(* Logix 5000 project; controller Commerford_topping_5477_V3 vendor 1 type 14 code 222 rev 33.11; software revision 33.02 *)

TASK MainTask (continuous, watchdog 500 ms) : MainProgram
TASK SafetyTask (periodic, rate 20 ms, priority 10, watchdog 20 ms, safety) : SafetyProgram
TASK Unit6_Topping_system (event, rate 10 ms, priority 10, watchdog 500 ms) : UN6_Object, UN6_EM1_Buffertank, UN6_EM2_Color_1, UN6_EM3_Color_2, UN6_EM4_Color_3, UN6_EM5_No_Color

MODULES
   Local : vendor 1 type 14 code 222 (5069 0, rev 33.11)
END_MODULES

TYPE Descriptor :   // is used for recipes
STRUCT
   Value : REAL;   // Parameter Values
END_STRUCT
END_TYPE

TYPE EquipmentModule :   // EquipmentModule
STRUCT
   Selected : BOOL;   // EquipmentModule is active
   State_in : DINT;   // EM State request
   State_out : DINT;   // EM State complete
   Current_Action : STRING_32;   // Contains information about current action of equipment module
   Force_Stop : BOOL;   // Sets the statemodel to Stopping
   Force_Abort : BOOL;   // Sets the statemodel to Aborting
   Suspend_Trigger : BOOL;   // Requests a Suspending state
   Reset_Signal : BOOL;   // Reset for entire EM, this will be done by 1. Resetting 2. Clearing 3. HMI_Reset
   Faulted : BOOL;   // EquipmentModule is faulted locally
   CM_Force_Stop : BOOL;   // Sets the statemodel to Stopping, ONLY USED BY CM AOI. DO NOT USE OTHERWISE!!
   CM_Force_Abort : BOOL;   // Sets the statemodel to Aborting, ONLY USED BY CM AOI. DO NOT USE OTHERWISE!!
   _SEQ : EquipmentModule_SEQ;
END_STRUCT
END_TYPE

TYPE EquipmentModule_SEQ :
STRUCT
   Clearing : INT;   // Step nummer
   Activating : INT;   // Step nummer
   Deactivating : INT;   // Step nummer
   Aborting : INT;   // Step nummer
   Resetting : INT;   // Step nummer
END_STRUCT
END_TYPE

TYPE MasterRecipeSelect :
STRUCT
   Recipe : STRING_476;
   SelectedRecipeNum : DINT;
   SelectedProces : DINT;
   RunRecipe : BOOL;   // Set to true to download recipe to proces
   Process : STRING_476;
END_STRUCT
END_TYPE

TYPE Packml_States :   // Enum for packml states
STRUCT
   Aborting : BOOL;   // Packml state
   Aborted : BOOL;   // Packml state
   Clearing : BOOL;   // Packml state
   Stopping : BOOL;   // Packml state
   Stopped : BOOL;   // Packml state
   Resetting : BOOL;   // Packml state
   Idle : BOOL;   // Packml state
   Starting : BOOL;   // Packml state
   Execute : BOOL;   // Packml state
   Holding : BOOL;   // Packml state
   Held : BOOL;   // Packml state
   Unholding : BOOL;   // Packml state
   Suspending : BOOL;   // Packml state
   Suspended : BOOL;   // Packml state
   Unsuspending : BOOL;   // Packml state
   Completing : BOOL;   // Packml state
   Complete : BOOL;   // Packml state
END_STRUCT
END_TYPE

TYPE PLMs :   // Status tags are used to describe the operation of the unit machine. Status tags include state commands which describe the state transitions in the Base State Model. The status tags also include parameters and process variables which describe how the machine operates.
STRUCT
   UnitModeCurrent : DINT;   // Unit Mode in Current Use
   UnitModeRequested : BOOL;   // Requested Unit Mode Change
   UnitModeChangeInProcess : BOOL;   // Requested Unit Mode Change in Process
   StateCurrent : DINT;   // Current State Number
   StateRequested : DINT;   // Target State.
   StateChangeInProcess : BOOL;   // State Change in Process.
   MachSpeed : REAL;   // Current Machine Speed
   CurMachSpeed : REAL;   // Current Machine Speed in Primary Packages/Minute
   MaterialInterlock : BOOL;   // Materials Ready
   UnitFaulted : BOOL;   // Machine is faulted
END_STRUCT
END_TYPE

TYPE PMLc :   // Command tags are used to control the operation of the unit machine. Command tags include unit state commands which control the state transitions in the Base State Model.
STRUCT
   UnitMode : DINT;   // This value is predefined by the user/OEM, and are the desired unit modes of the machine.
   UnitModeChangeRequest : BOOL;   // When a unit mode request takes place a numerical value must be present in the Command.UnitMode tag to change the unit mode.
   MaterialsInterlocks : BOOL;
   CntrlCmd : DINT;   // 0 Undefined 1 Reset 2 Start 3 Stop 4 Hold 5 Unhold 6 Suspend 7 Unsuspend 8 Abort 9 Clear
   CmdChangeRequest : BOOL;   // This CmdChangeRequest bit will command the machine to proceed to change the state to the target state. The tag can be used to condition when a change of state can occur. The target state will be one of the states in the base state model.
END_STRUCT
END_TYPE

TYPE Process_Status :
STRUCT
   Running : BOOL;   // Phase is executing Running logic
   Complete : BOOL;   // Phase is completed, waiting for reset command
   Held : BOOL;   // Phase is held, waiting for Restart command
   Idle : BOOL;   // Phase is Idle, waiting for Start command
   Resetting : BOOL;   // Phase is executing Resetting logic
   Stopped : BOOL;   // Phase is Stopped, waiting for Reset command
   Aborted : BOOL;   // Phase is Aborted, waiting for Reset command
   Aborting : BOOL;   // Phase is executing Aborting logic
   Stopping : BOOL;   // Phase is executing Stopping logic
   Holding : BOOL;   // Phase is executing Holding logic
   Restarting : BOOL;   // Phase is executing Restarting logic
   Ready : BOOL;   // Phase Completed, phase is ready to recieve new commands
END_STRUCT
END_TYPE

TYPE ProcessModule :
STRUCT
   Selected : BOOL;   // Process is active
   State_in : DINT;   // Process State request
   State_out : DINT;   // Process State complete
   Force_Stop : BOOL;   // Sets the statemodel to Stopping
   Force_Abort : BOOL;   // Sets the statemodel to Aborting
   Suspend_Trigger : BOOL;   // Requests a Suspending state
   Faulted : BOOL;   // Process is faulted locally
   Status : Process_Status;   // Status of process
END_STRUCT
END_TYPE

TYPE StateCurrentTime_array :   // sub array
STRUCT
   Mode : DINT[18];
END_STRUCT
END_TYPE

TYPE STRING_476 :   // Max chars HMI supports.
STRUCT
   LEN : DINT;
   DATA : SINT[476];
END_STRUCT
END_TYPE

ADD_ON_INSTRUCTION EquipmentModule_Link   (* revision 1.1, vendor WPI *)
// Revision note:
// 1.1 - CM faults reset
VAR_IN_OUT
   PackML : ISA_TR_88_00_02; {required}
   EquipmentModule : EquipmentModule; {required}
   bStateTransitions : DINT[32]; {required}
END_VAR
VAR_INPUT
   EM_ID : DINT; {required}
   Select : BOOL; {visible}   // Selecting EM will incuding in Unit state transitions
END_VAR
VAR_OUTPUT
   Sts_EM_Selected : BOOL; {access Read Only, visible}
   OwnershipFault : BOOL; {access Read Only, visible}
   Sts_Clearing_PC : BOOL; {access Read Only, visible}
   Sts_Starting_PC : BOOL; {access Read Only, visible}
   Sts_Executing : BOOL; {access Read Only, visible}
   Sts_Stopping_PC : BOOL; {access Read Only, visible}
   Sts_Aborting_PC : BOOL; {access Read Only, visible}
   Sts_Holding_PC : BOOL; {access Read Only, visible}
   Sts_Unholding_PC : BOOL; {access Read Only, visible}
   Sts_Suspending_PC : BOOL; {access Read Only, visible}
   Sts_Resetting_PC : BOOL; {access Read Only, visible}
   Sts_Unsuspending_PC : BOOL; {access Read Only, visible}
   Sts_Completing_PC : BOOL; {access Read Only, visible}
   Sts_SuspendTrigger : BOOL; {access Read Only, visible}
   Sts_Faulted : BOOL; {access Read Only, visible}
   Sts_Force_Stop : BOOL; {access Read Only, visible}
   Sts_Force_Abort : BOOL; {access Read Only, visible}
END_VAR
VAR
   AsignOwnership : BOOL; {access None}
   UnasignOwnership : BOOL; {access None}
END_VAR

ROUTINE Logic   (* ladder *)
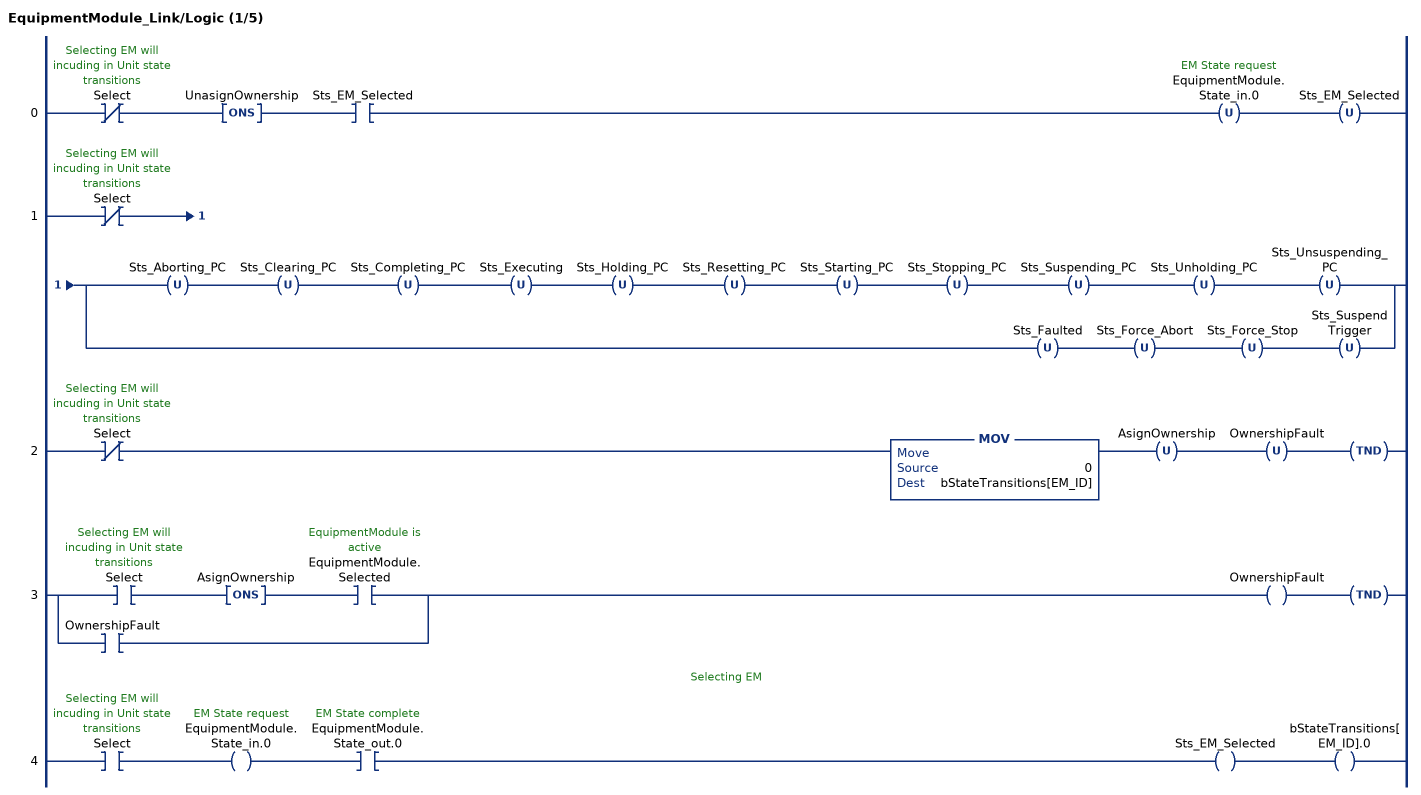
   0: XIO(Select)ONS(UnasignOwnership)XIC(Sts_EM_Selected)OTU(EquipmentModule.State_in.0)OTU(Sts_EM_Selected);
   1: XIO(Select)[OTU(Sts_Aborting_PC) OTU(Sts_Clearing_PC) OTU(Sts_Completing_PC) OTU(Sts_Executing) OTU(Sts_Holding_PC) OTU(Sts_Resetting_PC) OTU(Sts_Starting_PC) OTU(Sts_Stopping_PC) OTU(Sts_Suspending_PC) OTU(Sts_Unholding_PC) OTU(Sts_Unsuspending_PC) ,OTU(Sts_Faulted) OTU(Sts_Force_Abort) OTU(Sts_Force_Stop) OTU(Sts_SuspendTrigger) ];
   2: XIO(Select)MOV(0,bStateTransitions[EM_ID])OTU(AsignOwnership)OTU(OwnershipFault)TND();
   3: [XIC(Select) ONS(AsignOwnership) XIC(EquipmentModule.Selected) ,XIC(OwnershipFault) ]OTE(OwnershipFault)TND();
   // Selecting EM
   4: XIC(Select)OTE(EquipmentModule.State_in.0)XIC(EquipmentModule.State_out.0)OTE(Sts_EM_Selected)OTE(bStateTransitions[EM_ID].0);
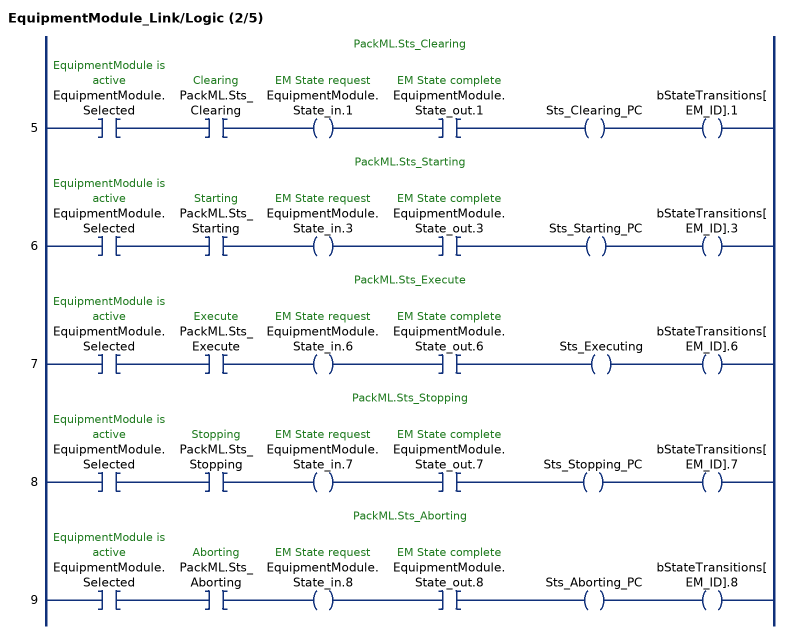
   // PackML.Sts_Clearing
   5: XIC(EquipmentModule.Selected)XIC(PackML.Sts_Clearing)OTE(EquipmentModule.State_in.1)XIC(EquipmentModule.State_out.1)OTE(Sts_Clearing_PC)OTE(bStateTransitions[EM_ID].1);
   // PackML.Sts_Starting
   6: XIC(EquipmentModule.Selected)XIC(PackML.Sts_Starting)OTE(EquipmentModule.State_in.3)XIC(EquipmentModule.State_out.3)OTE(Sts_Starting_PC)OTE(bStateTransitions[EM_ID].3);
   // PackML.Sts_Execute
   7: XIC(EquipmentModule.Selected)XIC(PackML.Sts_Execute)OTE(EquipmentModule.State_in.6)XIC(EquipmentModule.State_out.6)OTE(Sts_Executing)OTE(bStateTransitions[EM_ID].6);
   // PackML.Sts_Stopping
   8: XIC(EquipmentModule.Selected)XIC(PackML.Sts_Stopping)OTE(EquipmentModule.State_in.7)XIC(EquipmentModule.State_out.7)OTE(Sts_Stopping_PC)OTE(bStateTransitions[EM_ID].7);
   // PackML.Sts_Aborting
   9: XIC(EquipmentModule.Selected)XIC(PackML.Sts_Aborting)OTE(EquipmentModule.State_in.8)XIC(EquipmentModule.State_out.8)OTE(Sts_Aborting_PC)OTE(bStateTransitions[EM_ID].8);
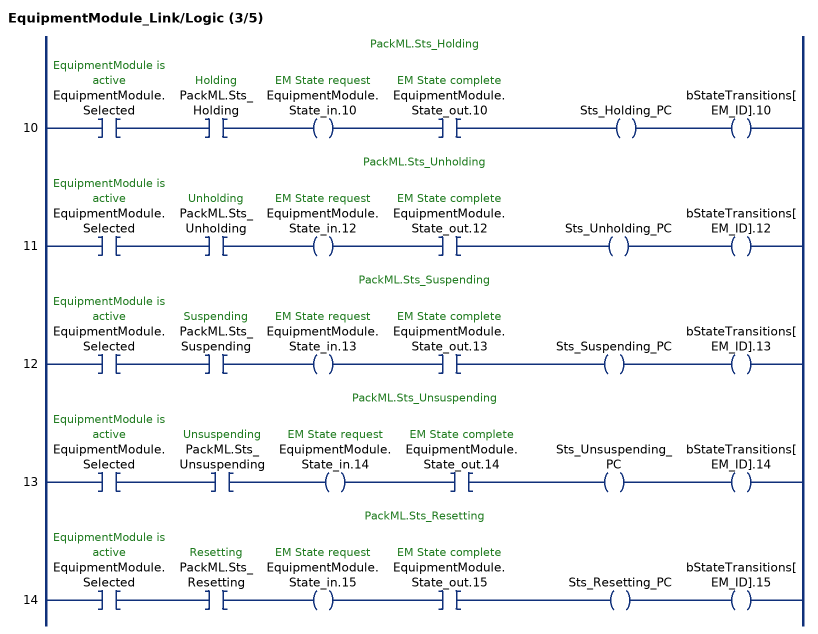
   // PackML.Sts_Holding
   10: XIC(EquipmentModule.Selected)XIC(PackML.Sts_Holding)OTE(EquipmentModule.State_in.10)XIC(EquipmentModule.State_out.10)OTE(Sts_Holding_PC)OTE(bStateTransitions[EM_ID].10);
   // PackML.Sts_Unholding
   11: XIC(EquipmentModule.Selected)XIC(PackML.Sts_Unholding)OTE(EquipmentModule.State_in.12)XIC(EquipmentModule.State_out.12)OTE(Sts_Unholding_PC)OTE(bStateTransitions[EM_ID].12);
   // PackML.Sts_Suspending
   12: XIC(EquipmentModule.Selected)XIC(PackML.Sts_Suspending)OTE(EquipmentModule.State_in.13)XIC(EquipmentModule.State_out.13)OTE(Sts_Suspending_PC)OTE(bStateTransitions[EM_ID].13);
   // PackML.Sts_Unsuspending
   13: XIC(EquipmentModule.Selected)XIC(PackML.Sts_Unsuspending)OTE(EquipmentModule.State_in.14)XIC(EquipmentModule.State_out.14)OTE(Sts_Unsuspending_PC)OTE(bStateTransitions[EM_ID].14);
   // PackML.Sts_Resetting
   14: XIC(EquipmentModule.Selected)XIC(PackML.Sts_Resetting)OTE(EquipmentModule.State_in.15)XIC(EquipmentModule.State_out.15)OTE(Sts_Resetting_PC)OTE(bStateTransitions[EM_ID].15);
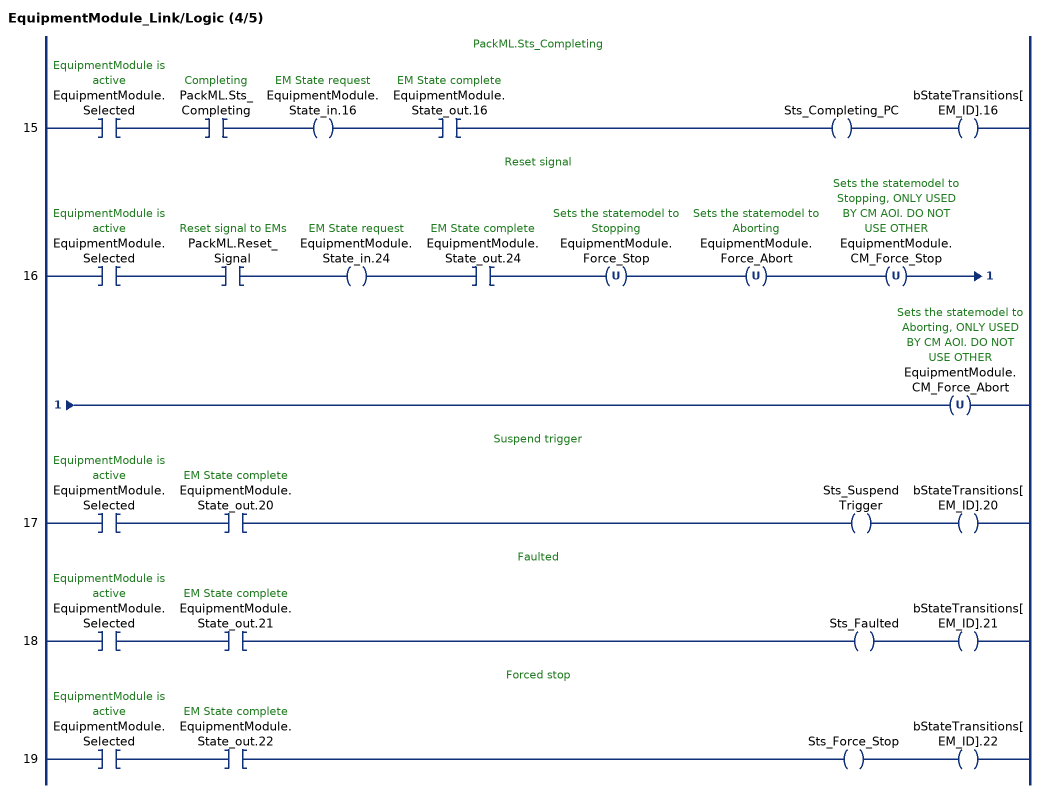
   // PackML.Sts_Completing
   15: XIC(EquipmentModule.Selected)XIC(PackML.Sts_Completing)OTE(EquipmentModule.State_in.16)XIC(EquipmentModule.State_out.16)OTE(Sts_Completing_PC)OTE(bStateTransitions[EM_ID].16);
   // Reset signal
   16: XIC(EquipmentModule.Selected)XIC(PackML.Reset_Signal)OTE(EquipmentModule.State_in.24)XIC(EquipmentModule.State_out.24)OTU(EquipmentModule.Force_Stop)OTU(EquipmentModule.Force_Abort)OTU(EquipmentModule.CM_Force_Stop)OTU(EquipmentModule.CM_Force_Abort);
   // Suspend trigger
   17: XIC(EquipmentModule.Selected)XIC(EquipmentModule.State_out.20)OTE(Sts_SuspendTrigger)OTE(bStateTransitions[EM_ID].20);
   // Faulted
   18: XIC(EquipmentModule.Selected)XIC(EquipmentModule.State_out.21)OTE(Sts_Faulted)OTE(bStateTransitions[EM_ID].21);
   // Forced stop
   19: XIC(EquipmentModule.Selected)XIC(EquipmentModule.State_out.22)OTE(Sts_Force_Stop)OTE(bStateTransitions[EM_ID].22);
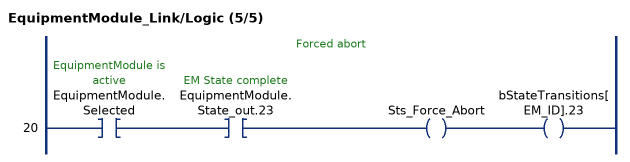
   // Forced abort
   20: XIC(EquipmentModule.Selected)XIC(EquipmentModule.State_out.23)OTE(Sts_Force_Abort)OTE(bStateTransitions[EM_ID].23);
END_ROUTINE
END_ADD_ON_INSTRUCTION

ADD_ON_INSTRUCTION ISA_TR_88_00_02   (* revision 1.2, ExecutePrescan *)
// Machine and Unit States:
// An Implementation Example of
// ISA-88
// Revision note:
// Processactive update
// Help:
// Read parameter list for documentation
VAR_IN_OUT
   PackTags : PACKMLv30; {required}
   EquipmentModules : DINT[32]; {required}
END_VAR
VAR_OUTPUT
   Sts_SC_Status : UDINT; {access Read Only, visible}
   Sts_Clearing : BOOL; {access Read Only, visible}   // Clearing
   Sts_Stopped : BOOL; {access Read Only, visible}   // Stopped
   Sts_Starting : BOOL; {access Read Only, visible}   // Starting
   Sts_Idle : BOOL; {access Read Only, visible}   // Idle
   Sts_Suspended : BOOL; {access Read Only, visible}   // Suspended
   Sts_Execute : BOOL; {access Read Only, visible}   // Execute
   Sts_Stopping : BOOL; {access Read Only, visible}   // Stopping
   Sts_Aborting : BOOL; {access Read Only, visible}   // Aborting
   Sts_Aborted : BOOL; {access Read Only, visible}   // Aborted
   Sts_Holding : BOOL; {access Read Only, visible}   // Holding
   Sts_Held : BOOL; {access Read Only, visible}   // Held
   Sts_Unholding : BOOL; {access Read Only, visible}   // Unholding
   Sts_Suspending : BOOL; {access Read Only, visible}   // Suspending
   Sts_Unsuspending : BOOL; {access Read Only, visible}   // Unsuspending
   Sts_Resetting : BOOL; {access Read Only, visible}   // Resetting
   Sts_Completing : BOOL; {access Read Only, visible}   // Completing
   Sts_Complete : BOOL; {access Read Only, visible}   // Complete
   Sts_Automatic : BOOL; {access Read Only, visible}   // Machine is in fully automatic mode
   Sts_Maintenance : BOOL; {access Read Only, visible}   // Machine is in Maintenance
   Sts_Manual : BOOL; {access Read Only, visible}   // Machine is in Manual
END_VAR
VAR_INPUT
   Process_Selected : SINT; {visible}   // Recipe number selects which PackTag.command.product[#] will be used.
END_VAR
VAR_OUTPUT
   Sts_MachineFaulted : BOOL; {access Read Only, visible}   // Machine recieved an fault trigger
END_VAR
VAR_INPUT
   HMI_Reset : BOOL;   // Common reset for all EMs
END_VAR
VAR_OUTPUT
   Sts_ProcessActive : BOOL; {access Read Only, visible}   // Machine is running a process.
   Reset_Signal : BOOL; {access Read Only}   // Reset signal to EMs
END_VAR
VAR_IN_OUT
   Processes : DINT[32]; {required}
   Cnf_EnableMachineStates : Packml_States; {required}
END_VAR
VAR
   MachineState : USINT := 255; {access None}   // Technical Report Equipment States: 1 Clearing 2 Stopped 3 Starting 4 Idle 5 Suspended 6 Execute 7 Stopping 8 Aborting 9 Aborted 10 Holding 11 Held 12 Unholding 13 Suspending 14 Unsuspending 15 Resetting 16 Completing 17 Complete
   wrk_compare_UDINT : UDINT := 65535; {access None}
   wrk_Aborting_to_Aborted : UDINT := 2#0000_0000_0000_0000_1111_1111_1111_1111; {access None}
   i : DINT; {access None}   // index num, only for local use. used for forloops
   Wrk_Aborting_to_Aborted_PC : BOOL; {access None}   // EquipmentModule(s) Aborting_to_Aborted Proces Complete
   FALSE : BOOL; {access None}   // always false
   TRUE : BOOL; {access None}   // always true
   wrk_Conversion : DINT; {access None}
   temp_sum : DINT; {access None}   // local storage
   wrk_Stopping_to_Stopped : UDINT; {access None}
   wrk_Starting_to_Execute : UDINT; {access None}
   wrk_Clearing_to_Stopped : UDINT; {access None}
   wrk_Holding_to_Held : UDINT; {access None}
   wrk_Unholding_to_Execute : UDINT; {access None}
   wrk_Suspending_to_Suspended : UDINT; {access None}
   wrk_Unsuspending_to_Execute : UDINT; {access None}
   wrk_Resetting_to_Idle : UDINT; {access None}
   wrk_Completing_to_Completed : UDINT; {access None}
   wrk_prev_state : DINT; {access None}   // local mem
   MachineMode : DINT; {access None}
   wrk_SwitchLayer_To_Maintenance : DINT; {access None}
   wrk_SwitchLayer_To_Manual : DINT; {access None}
   wrk_SwitchLayer_To_Automatic : DINT; {access None}
   k : DINT; {access None}   // nested index num
   ArraySize : DINT[5]; {access None}   // local array size
   wrk_RecipeNumber : DINT; {access None}   // local RecipeNum
   DEL_T_Refresh_PackTag_Status : FBD_TIMER; {access None}
   T_second_puls : FBD_TIMER; {access None}   // local timer for just 1 second
   T_Refresh_PackTag_Administration : FBD_TIMER; {access None}   // local timer
   wrk_DateTime : LINT; {access None}
   wrk_Execute_to_Completing : UDINT; {access None}
   T_ResetSignal_ON : FBD_TIMER; {access None}   // Local reset timer
   T_ResetSignal_OFF : FBD_TIMER; {access None}   // local reset timer
   T_ResetSignal_HMI : FBD_TIMER; {access None}   // reset timer from HMI
   StateHistory : StateHistory[10]; {access Read Only}
   debugProg : DINT; {access None}
   wrk_HandHalt : BOOL; {access None}   // machine is forced to stop by user
   Wrk_EM_Restting : UDINT; {access None}
   Wrk_Process_Restting : UDINT; {access None}
   Wrk_Process_Starting : UDINT; {access None}
   Wrk_Process_Completing : UDINT; {access None}
   Wrk_EM_Starting : UDINT; {access None}
   Wrk_EM_Completed : UDINT; {access None}
   Wrk_EM_Stopping : UDINT; {access None}
   Wrk_EM_Aborting : UDINT; {access None}
   Wrk_EM_Holding : UDINT; {access None}
   Wrk_EM_Unholding : UDINT; {access None}
   Wrk_EM_Suspending : UDINT; {access None}
   Wrk_EM_Unsuspending : UDINT; {access None}
   Wrk_Process_Stopping : UDINT; {access None}
   Wrk_Process_Aborting : UDINT; {access None}
   Wrk_processes_Holding : UDINT; {access None}
   Wrk_processes_Unholding : UDINT; {access None}
   Wrk_processes_Suspending : UDINT; {access None}
   Wrk_processes_Unsuspending : UDINT; {access None}
   Wrk_processes_Completed : UDINT; {access None}
   Wrk_EM_Clearing : UDINT; {access None}
   Wrk_Process_Clearing : UDINT; {access None}
END_VAR

ROUTINE Logic   (* structured text *)
// Machine and Unit States:
// An Implementation Example of
// ISA-88
   ////////////////////////////////////////////////////////////
   //   Copyright (c)
   //------------------------------------------------------------
   //   Routine: ISA_TR_88_00_02 - Logic
   //   Author: WPI\tom.reit
   //   Created: 2-11-2022
   //------------------------------------------------------------
   //   Description:
   //           Machine and Unit States:
   //           An Implementation Example of
   //           ISA-88
   //
   //
   //   History:
   //
   ////////////////////////////////////////////////////////////
   #region Macros / keywords
   	TRUE:=1;
   	FALSE:=0;
   	#region Second timer
   		if T_second_puls.DN then
   			T_second_puls.Reset:=TRUE;
   		else
   			T_second_puls.Reset:=FALSE;
   		end_if;
   		T_second_puls.TimerEnable	:=TRUE;
   		T_second_puls.PRE			:=1000;
   		TONR(T_second_puls);
   	#endregion
   	#region Reset timers
   	//On users request to reset or clear the machine there will be a resetSignal set for 50mS an it will be low for 100mS. once these timers are done, the machine will check feedback from EMs
   		T_ResetSignal_ON.TimerEnable	:=Sts_Clearing OR Sts_Resetting;											// once machine is in clearing or resetting or reset is pressed on HMI set reset for 50mS
   		T_ResetSignal_ON.PRE			:=50;																		// reset high time
   		T_ResetSignal_ON.Reset			:=(Sts_Stopped OR Sts_Aborted OR Sts_Idle) AND T_ResetSignal_OFF.DN;		// clear timer
   
   		T_ResetSignal_OFF.PRE			:=100;																		// time reset signal off
   		T_ResetSignal_OFF.TimerEnable	:=T_ResetSignal_ON.DN;														// start time off once time on is done.
   		T_ResetSignal_OFF.Reset			:=T_ResetSignal_OFF.DN AND NOT (Sts_Clearing OR Sts_Resetting);				// clear timer
   
   		T_ResetSignal_HMI.PRE			:=50;																		// time reset signal off
   		T_ResetSignal_HMI.TimerEnable	:=(HMI_Reset OR T_ResetSignal_HMI.TT);										// start time off once time on is done.
   		T_ResetSignal_HMI.Reset			:=T_ResetSignal_HMI.DN AND NOT HMI_Reset;															// clear timer
   
   		TONR(T_ResetSignal_ON);																						// timer object
   		TONR(T_ResetSignal_OFF);																					// timer object
   		TONR(T_ResetSignal_HMI);																					// timer object
   
   		if T_ResetSignal_ON.TT then
   			if NOT Reset_Signal then Reset_Signal:=TRUE; end_if;					// set reset signal for all EMs
   		end_if;
   		if T_ResetSignal_OFF.TT then
   			if Reset_Signal then Reset_Signal:=FALSE; end_if;						// unset reset signal for all EMs
   		end_if;
   
   		if T_ResetSignal_HMI.TT then
   			if NOT Reset_Signal then Reset_Signal:=TRUE; end_if;						// set reset signal for all EMs
   		end_if;
   		if T_ResetSignal_HMI.DN then
   			if Reset_Signal then Reset_Signal:=FALSE; end_if;						// set reset signal for all EMs
   			HMI_Reset:=FALSE;
   		end_if;
   	#endregion
   
   #endregion
   
   #region Machine States
   /*Discription
   A State transition is defined as a passage from one state to another. Transitions between
   states will occur as a result of a local, remote, or procedural State command.
   
   
   for the SC's we use the following bit manipulation run a forloop from 0 till max array size.
   each cycle of the forloop check if EMs_Status[i]Request_SC.XXXXX is true or false.
   
   since an bool can not be directly moved into an UDINT we do some clever calculations
   (1*2)^i OR (0*2)^i this will result into an DEC value based on the BIN bit num.
   
   forexample BIN the value is 1011 this is DEC 13 if we want to convert 1011 to an DEC value we cycle through each bit using an index num. so
   
   BIT value		Index num			Calculation			Result
   	1				0				(1*2)^0					1
   	0				1				(0*2)^1					0
   	1				2				(1*2)^2					4
   	1				3				(1*2)^3					8
   
   	now we sum up result which is 1+0+4+8 = 13.
   	this way we have converted an array of bools into an UDINT. Now we can compare an UDINT with an compare value(all 32 bits to TRUE)
   */
   #region Switch layer to Maintenance
   	case wrk_SwitchLayer_To_Maintenance of
   		0: // check for request
   			if PackTags.Command.UnitMode = 2 AND PackTags.Command.UnitModeChangeRequest then 									// request from HMI
   				PackTags.Status.UnitModeRequested		:=TRUE;						// request mode
   				PackTags.Status.UnitModeChangeInProcess	:=TRUE;						// changing mode
   				wrk_SwitchLayer_To_Maintenance			:=1;						// Set to next step
   			end_if;
   		1: // Set all modules in request mode
   			wrk_SwitchLayer_To_Maintenance:=2;										// set to next step
   		2: // Set unit to new mode.
   			PackTags.Status.UnitModeChangeInProcess	:=FALSE;						// changing mode done
   			PackTags.Status.UnitModeRequested		:=FALSE;						// request mode
   			PackTags.Command.UnitMode				:=0;							// unlatch signal on HMI as feedback.
   			MachineMode								:=2;							// Set machine in other layer.
   			wrk_SwitchLayer_To_Maintenance			:=0;							// reset statemodel
   		else // undefined state
   			wrk_SwitchLayer_To_Maintenance:=0;
   	end_case;
   	if wrk_SwitchLayer_To_Maintenance <> 0 AND NOT (PackTags.Command.UnitMode=2) then
   		wrk_SwitchLayer_To_Maintenance:=0; 											// reset request once signal is set back to 0 and machine did not switch layer.
   	end_if;
   #endregion
   
   #region Switch layer to Manual
   	case wrk_SwitchLayer_To_Manual of
   		0: // check for request
   			if PackTags.Command.UnitMode = 3 AND PackTags.Command.UnitModeChangeRequest then 								// request from HMI
   				PackTags.Status.UnitModeRequested		:=TRUE;						// request mode
   				PackTags.Status.UnitModeChangeInProcess	:=TRUE;						// changing mode
   				wrk_SwitchLayer_To_Manual				:=1;						// Set to next step
   			end_if;
   		1: // Set all modules in request mode
   			wrk_SwitchLayer_To_Manual:=2;											// set to next step
   		2: // Set unit to new mode.
   			PackTags.Status.UnitModeChangeInProcess	:=FALSE;						// changing mode done
   			PackTags.Status.UnitModeRequested		:=FALSE;						// request mode
   			PackTags.Command.UnitMode				:=0;							// unlatch signal on HMI as feedback.
   			MachineMode								:=3;							// Set machine in other layer.
   			wrk_SwitchLayer_To_Manual				:=0;							// reset statemodel
   		else // undefined state
   			wrk_SwitchLayer_To_Manual:=0;
   	end_case;
   	if wrk_SwitchLayer_To_Manual <> 0 AND NOT (PackTags.Command.UnitMode=3) then
   		wrk_SwitchLayer_To_Manual:=0; 											// reset request once signal is set back to 0 and machine did not switch layer.
   	end_if;
   #endregion
   
   #region Switch layer to Automatic
   	case wrk_SwitchLayer_To_Automatic of
   		0: // check for request
   			if PackTags.Command.UnitMode=1 AND PackTags.Command.UnitModeChangeRequest then 								// request from HMI
   				PackTags.Status.UnitModeRequested		:=TRUE;						// request mode
   				PackTags.Status.UnitModeChangeInProcess	:=TRUE;						// changing mode
   				wrk_SwitchLayer_To_Automatic			:=1;						// Set to next step
   			end_if;
   		1: // Set all modules in request mode
   			wrk_SwitchLayer_To_Automatic:=2;											// set to next step
   		2: // Set unit to new mode.
   			PackTags.Status.UnitModeChangeInProcess		:=FALSE;						// changing mode done
   			PackTags.Status.UnitModeRequested			:=FALSE;						// request mode
   			PackTags.Command.UnitMode					:=0;							// unlatch signal on HMI as feedback.
   			MachineMode									:=1;							// Set machine in other layer.
   			wrk_SwitchLayer_To_Automatic				:=0;							// reset statemodel
   		else // undefined state
   			wrk_SwitchLayer_To_Automatic:=0;
   	end_case;
   	if wrk_SwitchLayer_To_Automatic <> 0 AND NOT (PackTags.Command.UnitMode=1) then
   		wrk_SwitchLayer_To_Automatic:=0; 											// reset request once signal is set back to 0 and machine did not switch layer.
   	end_if;
   #endregion
   
   case MachineMode of
   	0:  /*************************		Undefined		*****************************	*/
   		MachineMode:=1;
   
   		PackTags.Status.UnitModeCurrent:=0;
   	1: 	/*************************		Automatic		*****************************	*/
   		Sts_Automatic		:=TRUE;
   		Sts_Maintenance		:=FALSE;
   		Sts_Manual			:=FALSE;
   
   		PackTags.Status.UnitModeCurrent:=1;
   	2: 	/*************************		Maintenance		*****************************	*/
   		Sts_Automatic		:=FALSE;
   		Sts_Maintenance		:=TRUE;
   		Sts_Manual			:=FALSE;
   
   		PackTags.Status.UnitModeCurrent:=2;
   	3: 	/*************************		Manual			*****************************	*/
   		Sts_Automatic		:=FALSE;
   		Sts_Maintenance		:=FALSE;
   		Sts_Manual			:=TRUE;
   
   		PackTags.Status.UnitModeCurrent:=3;
   	4: 	/*************************		Spare			*****************************	*/
   	5: 	/*************************		Spare			*****************************	*/
   	6: 	/*************************		Spare			*****************************	*/
   	7: 	/*************************		Spare			*****************************	*/
   	8: 	/*************************		Spare			*****************************	*/
   	9: 	/*************************		Spare			*****************************	*/
   	10: /*************************		Spare			*****************************	*/
   	11: /*************************		Spare			*****************************	*/
   	12: /*************************		Spare			*****************************	*/
   	13: /*************************		Spare			*****************************	*/
   	14: /*************************		Spare			*****************************	*/
   	15: /*************************		Spare			*****************************	*/
   	16: /*************************		UserDefined1	*****************************	*/
   	17: /*************************		UserDefined2	*****************************	*/
   
   	else
   		MachineMode:=0; // undefined state
   end_case;
   #region Machine active states
   	/*
   	Programmer can set states that will be active on unit. if not set, Packml will ignore them as if they are transition OK
   	thefor passing through them without setting underlaying equipment in that state
   	*/
   
   	/* Preset states that ALWAYS have to be included */
   	Cnf_EnableMachineStates.Aborted		:=TRUE;
   	Cnf_EnableMachineStates.Aborting	:=TRUE;
   
   	Cnf_EnableMachineStates.Execute		:=TRUE;
   	Cnf_EnableMachineStates.Stopped		:=TRUE;
   #endregion
   
   
   
   
   
   
   
   	case MachineState of
   		1: 	/******************************************************		Clearing	******************************************************/
   			#region Check EquipmentModule StateControl (SC)
   			temp_sum:=0;
   			PackTags.Status.StateRequested:=2;											// request Stopped state.
   			wrk_HandHalt:=0;
   			if Cnf_EnableMachineStates.Clearing then
   				if T_ResetSignal_OFF.DN then											// wait for reset seq for unit
   					for i := 0 to 31 do													// scan from 0 till max array size
   						if EquipmentModules[i].0 then									// check if EquipmentModule is selected
   							if EquipmentModules[i].1 then								// Feedback from equipmentmodule
   								wrk_Clearing_to_Stopped:=(1*2**i)+temp_sum; 			// state is true. convert binary to dec value. sum= bits *2 ^ i. See https://flexiple.com/developers/decimal-to-binary-conversion
   						 	else
   								wrk_Clearing_to_Stopped:=(0*2**i)+temp_sum; 			// state is false. convert binary to dec value. sum= bits *2 ^ i. See https://flexiple.com/developers/decimal-to-binary-conversion
   							end_if;
   						end_if;
   						if NOT EquipmentModules[i].0 then wrk_Clearing_to_Stopped:=(1*2**i)+temp_sum; end_if; // module is not enabled. therfor state is always true.
   						temp_sum:=wrk_Clearing_to_Stopped;
   					end_for;
   					Sts_SC_Status:=wrk_Clearing_to_Stopped;
   					Wrk_EM_Clearing:=wrk_Clearing_to_Stopped;
   
   
   					temp_sum:=0;
   					for i := 0 to 31 do													// scan from 0 till max array size
   						if Processes[i].0 then									// check if EquipmentModule is selected
   							if Processes[i].1 then								// Feedback from equipmentmodule
   								wrk_Clearing_to_Stopped:=(1*2**i)+temp_sum; 			// state is true. convert binary to dec value. sum= bits *2 ^ i. See https://flexiple.com/developers/decimal-to-binary-conversion
   						 	else
   								wrk_Clearing_to_Stopped:=(0*2**i)+temp_sum; 			// state is false. convert binary to dec value. sum= bits *2 ^ i. See https://flexiple.com/developers/decimal-to-binary-conversion
   							end_if;
   						end_if;
   						if NOT Processes[i].0 then wrk_Clearing_to_Stopped:=(1*2**i)+temp_sum; end_if; // module is not enabled. therfor state is always true.
   						temp_sum:=wrk_Clearing_to_Stopped;
   					end_for;
   					Wrk_Process_Clearing:=wrk_Clearing_to_Stopped;
   					if (Wrk_EM_Clearing = wrk_compare_UDINT) AND (Wrk_Process_Clearing = wrk_compare_UDINT) then
   						Sts_MachineFaulted:=FALSE;										// Set machine faulted to false.
   						MachineState:=2;												//	move unit to Stopped.
   					end_if;
   				end_if;
   			else
   				MachineState:=2;
   			end_if;
   			#endregion
   
   
   		2:	/******************************************************		Stopped		******************************************************/
   			wrk_Clearing_to_Stopped	:=0; 											// clear old mem, since state was succesful.
   
   			if Cnf_EnableMachineStates.Stopped then
   				if PackTags.Command.CntrlCmd = 1 AND PackTags.Command.CmdChangeRequest then	//	The tag holds the value of the command that provides the state command to drive a state change in the Base State Model
   					PackTags.Status.StateRequested:=15;									//  request Resetting state.
   					MachineState	:=	15;												// 	move to resetting
   					PackTags.Command.CmdChangeRequest:=0;								//  accept request and set signal back low.
   				end_if;
   			else
   				PackTags.Status.StateRequested	:=	15;
   				MachineState					:=	15;
   			end_if;
   
   
   
   		3:	/******************************************************		Starting	******************************************************/
   			#region Check EquipmentModule StateControl (SC)
   			temp_sum:=0;
   
   			PackTags.Status.StateRequested:=6;										// request Execute state.
   			if Cnf_EnableMachineStates.Starting then
   				for i := 0 to 31 do										// scan from 0 till max array size
   					if EquipmentModules[i].0 then									// check if EquipmentModule is selected
   						if EquipmentModules[i].3 then		// Feedback from equipmentmodule
   							wrk_Starting_to_Execute:=(1*2**i)+temp_sum; 			// convert binary to dec value. sum= bits *2 ^ i. See https://flexiple.com/developers/decimal-to-binary-conversion
   					 	else
   							wrk_Starting_to_Execute:=(0*2**i)+temp_sum; 			// convert binary to dec value. sum= bits *2 ^ i. See https://flexiple.com/developers/decimal-to-binary-conversion
   						end_if;
   					end_if;
   					if NOT EquipmentModules[i].0 then wrk_Starting_to_Execute:=(1*2**i)+temp_sum; end_if; // module is not enabled. therfor state is always true.
   					temp_sum:=wrk_Starting_to_Execute;
   				end_for;
   				Sts_SC_Status:=wrk_Starting_to_Execute;
   				Wrk_EM_Starting:=wrk_Starting_to_Execute;
   				temp_sum:=0;
   				for i := 0 to 31 do										// scan from 0 till max array size
   					if Processes[i].0 then									// check if EquipmentModule is selected
   						if Processes[i].3 then			// Feedback from equipmentmodule
   							wrk_Starting_to_Execute:=(1*2**i)+temp_sum; 				// convert binary to dec value. sum= bits *2 ^ i. See https://flexiple.com/developers/decimal-to-binary-conversion
   					 	else
   							wrk_Starting_to_Execute:=(0*2**i)+temp_sum; 				// convert binary to dec value. sum= bits *2 ^ i. See https://flexiple.com/developers/decimal-to-binary-conversion
   						end_if;
   					end_if;
   					if NOT Processes[i].0 then wrk_Starting_to_Execute:=(1*2**i)+temp_sum; end_if; // module is not enabled. therfor state is always true.
   					temp_sum:=wrk_Starting_to_Execute;
   				end_for;
   				Wrk_Process_Starting:=wrk_Starting_to_Execute;
   				if (Wrk_EM_Starting = wrk_compare_UDINT) AND (Wrk_Process_Starting = wrk_compare_UDINT) then
   					MachineState:=6;												// move unit to Execute.
   				end_if;
   			else
   				MachineState:=6;
   			end_if;
   			#endregion
   
   
   
   		4:	/******************************************************		Idle		******************************************************/
   			wrk_Resetting_to_Idle	:=0; 											// clear old mem, since state was succesful.
   			Sts_MachineFaulted		:=FALSE;										// Set machine faulted to false.
   			if Cnf_EnableMachineStates.Idle then
   				if PackTags.Command.CntrlCmd = 2 AND PackTags.Command.CmdChangeRequest then //	The tag holds the value of the command that provides the state command to drive a state change in the Base State Model
   					PackTags.Status.StateRequested:=3;									// request Starting state.
   					MachineState:=3;													// move to starting
   					PackTags.Command.CmdChangeRequest:=0;								//  accept request and set signal back low.
   				end_if;
   			else
   					PackTags.Status.StateRequested:=3;									// request Starting state.
   					MachineState:=3;													// move to starting
   			end_if;
   
   
   
   		5:	/******************************************************		Suspended	******************************************************/
   			wrk_Suspending_to_Suspended	:=0; 										// clear old mem, since state was succesful.
   			if Cnf_EnableMachineStates.Suspended then
   				if PackTags.Command.CntrlCmd = 7 AND PackTags.Command.CmdChangeRequest then //	The tag holds the value of the command that provides the state command to drive a state change in the Base State Model
   					PackTags.Status.StateRequested:=14;									// request UnSuspend state.
   					MachineState:=14;													// move to unsuspending
   					PackTags.Command.CmdChangeRequest:=0;								//  accept request and set signal back low.
   				end_if;
   			else
   				PackTags.Status.StateRequested:=14;									// request UnSuspend state.
   				MachineState:=14;													// move to unsuspending
   			end_if;
   
   
   
   		6:	/******************************************************		Execute		******************************************************/
   			wrk_Starting_to_Execute		:=0; 										// clear old mem, since state was succesful.
   			wrk_Unholding_to_Execute	:=0; 										// clear old mem, since state was succesful.
   			wrk_Unsuspending_to_Execute	:=0; 										// clear old mem, since state was succesful.
   
   			#region Holding request
   				if Cnf_EnableMachineStates.Holding then
   					if PackTags.Command.CntrlCmd = 4 AND PackTags.Command.CmdChangeRequest then	// The tag holds the value of the command that provides the state command to drive a state change in the Base State Model
   						PackTags.Status.StateRequested:=10;									// request Holding state.
   						MachineState:=10;													// move to holding
   						PackTags.Command.CmdChangeRequest:=0;								//  accept request and set signal back low.
   					end_if;
   				else
   					if PackTags.Command.CntrlCmd = 4 AND PackTags.Command.CmdChangeRequest then
   						MachineState:=11;												// move directly to Held.
   						PackTags.Command.CmdChangeRequest:=0;							//  accept request and set signal back low.
   					end_if;
   				end_if;
   			#endregion
   			#region Suspending request
   				if Cnf_EnableMachineStates.Suspending then
   					if PackTags.Command.CntrlCmd = 6 AND PackTags.Command.CmdChangeRequest then // The tag holds the value of the command that provides the state command to drive a state change in the Base State Model
   						PackTags.Status.StateRequested:=13;									// request Suspending state.
   						MachineState:=13;													// move to suspending
   						PackTags.Command.CmdChangeRequest:=0;								//  accept request and set signal back low.
   					end_if;
   				else
   					if PackTags.Command.CntrlCmd = 6 AND PackTags.Command.CmdChangeRequest then // The tag holds the value of the command that provides the state command to drive a state change in the Base State Model
   						MachineState:=5;												// move directly to Suspended.
   						PackTags.Command.CmdChangeRequest:=0;							//  accept request and set signal back low.
   					end_if;
   				end_if;
   			#endregion
   			#region Completing request
   				if Cnf_EnableMachineStates.Completing then
   					if PackTags.Command.CntrlCmd = 10 AND PackTags.Command.CmdChangeRequest then	// The tag holds the value of the command that provides the state command to drive a state change in the Base State Model
   						PackTags.Status.StateRequested:=16;									// request Completing state.
   						MachineState:=16;													// move to Completing
   						PackTags.Command.CmdChangeRequest:=0;								//  accept request and set signal back low.
   					end_if;
   				else
   					if PackTags.Command.CntrlCmd = 10 AND PackTags.Command.CmdChangeRequest then	// The tag holds the value of the command that provides the state command to drive a state change in the Base State Model
   						MachineState:=17;												// move directly to Complete.
   						PackTags.Command.CmdChangeRequest:=0;							//  accept request and set signal back low.
   					end_if;
   				end_if;
   			#endregion
   
   			#region Check EquipmentModule StateControl (SC)
   			temp_sum:=0;
   				for i := 0 to 31 do										// scan from 0 till max array size
   					if EquipmentModules[i].0 then									// check if EquipmentModule is selected
   						if EquipmentModules[i].6 then		// Feedback from equipmentmodule
   							wrk_Execute_to_Completing:=(1*2**i)+temp_sum; 			// convert binary to dec value. sum= bits *2 ^ i. See https://flexiple.com/developers/decimal-to-binary-conversion
   					 	else
   							wrk_Execute_to_Completing:=(0*2**i)+temp_sum; 			// convert binary to dec value. sum= bits *2 ^ i. See https://flexiple.com/developers/decimal-to-binary-conversion
   						end_if;
   					end_if;
   					if NOT EquipmentModules[i].0 then wrk_Execute_to_Completing:=(1*2**i)+temp_sum; end_if; // module is not enabled. therfor state is always true.
   					temp_sum:=wrk_Execute_to_Completing;
   				end_for;
   				Sts_SC_Status:=wrk_Execute_to_Completing;
   				Wrk_EM_Completed:=wrk_Execute_to_Completing;
   				temp_sum:=0;
   					for i := 0 to 31 do										// scan from 0 till max array size
   						if Processes[i].0 then									// check if EquipmentModule is selected
   							if Processes[i].6 then			// Feedback from equipmentmodule
   								wrk_Execute_to_Completing:=(1*2**i)+temp_sum; 				// convert binary to dec value. sum= bits *2 ^ i. See https://flexiple.com/developers/decimal-to-binary-conversion
   						 	else
   								wrk_Execute_to_Completing:=(0*2**i)+temp_sum; 				// convert binary to dec value. sum= bits *2 ^ i. See https://flexiple.com/developers/decimal-to-binary-conversion
   							end_if;
   						end_if;
   						if NOT Processes[i].0 then wrk_Execute_to_Completing:=(1*2**i)+temp_sum; end_if; // module is not enabled. therfor state is always true.
   						temp_sum:=wrk_Execute_to_Completing;
   					end_for;
   					Wrk_Process_Completing:=wrk_Execute_to_Completing;
   				if (Wrk_EM_Completed = wrk_compare_UDINT) AND (Wrk_Process_Completing = wrk_compare_UDINT) then
   					if Cnf_EnableMachineStates.Completing then
   						MachineState:=16;												// move unit to Completing.
   					else
   						MachineState:=17;												// move unit to Completing.
   					end_if;
   				end_if;
   			#endregion
   
   
   
   		7:	/******************************************************		Stopping	******************************************************/
   			#region Check EquipmentModule StateControl (SC)
   			temp_sum:=0;
   
   			PackTags.Status.StateRequested:=2;										// request Stopped state.
   
   			if Cnf_EnableMachineStates.Stopping then
   				for i := 0 to 31 do										// scan from 0 till max array size
   					if EquipmentModules[i].0 then									// check if EquipmentModule is selected
   						if EquipmentModules[i].7 then		// Feedback from equipmentmodule
   							wrk_Stopping_to_Stopped:=(1*2**i)+temp_sum; 			// convert binary to dec value. sum= bits *2 ^ i. See https://flexiple.com/developers/decimal-to-binary-conversion
   					 	else
   							wrk_Stopping_to_Stopped:=(0*2**i)+temp_sum; 			// convert binary to dec value. sum= bits *2 ^ i. See https://flexiple.com/developers/decimal-to-binary-conversion
   						end_if;
   					end_if;
   					if NOT EquipmentModules[i].0 then wrk_Stopping_to_Stopped:=(1*2**i)+temp_sum; end_if; // module is not enabled. therfor state is always true.
   					temp_sum:=wrk_Stopping_to_Stopped;
   				end_for;
   				Sts_SC_Status:=wrk_Stopping_to_Stopped;
   				Wrk_EM_Stopping:=wrk_Stopping_to_Stopped;
   
   				temp_sum:=0;
   				for i := 0 to 31 do										// scan from 0 till max array size
   					if Processes[i].0 then									// check if EquipmentModule is selected
   						if Processes[i].7 then		// Feedback from equipmentmodule
   							wrk_Stopping_to_Stopped:=(1*2**i)+temp_sum; 			// convert binary to dec value. sum= bits *2 ^ i. See https://flexiple.com/developers/decimal-to-binary-conversion
   					 	else
   							wrk_Stopping_to_Stopped:=(0*2**i)+temp_sum; 			// convert binary to dec value. sum= bits *2 ^ i. See https://flexiple.com/developers/decimal-to-binary-conversion
   						end_if;
   					end_if;
   					if NOT Processes[i].0 then wrk_Stopping_to_Stopped:=(1*2**i)+temp_sum; end_if; // module is not enabled. therfor state is always true.
   					temp_sum:=wrk_Stopping_to_Stopped;
   				end_for;
   				Wrk_Process_Stopping:=wrk_Stopping_to_Stopped;
   
   				if (Wrk_EM_Stopping = wrk_compare_UDINT) AND (Wrk_Process_Stopping = wrk_compare_UDINT) then
   					MachineState:=2;												// move unit to Stopped.
   				end_if;
   			else
   				MachineState:=2;
   			end_if;
   			#endregion
   
   
   
   		8:	/******************************************************		Aborting	******************************************************/
   			#region Check EquipmentModule StateControl (SC)
   			temp_sum:=0;
   
   			PackTags.Status.StateRequested:=9;										// request Aborted state.
   			if Cnf_EnableMachineStates.Aborting then
   				for i := 0 to 31 do										// scan from 0 till max array size
   					if EquipmentModules[i].0 then									// check if EquipmentModule is selected
   						if EquipmentModules[i].8 then		// Feedback from equipmentmodule
   							wrk_Aborting_to_Aborted:=(1*2**i)+temp_sum; 			// convert binary to dec value. sum= bits *2 ^ i. See https://flexiple.com/developers/decimal-to-binary-conversion
   					 	else
   							wrk_Aborting_to_Aborted:=(0*2**i)+temp_sum; 			// convert binary to dec value. sum= bits *2 ^ i. See https://flexiple.com/developers/decimal-to-binary-conversion
   						end_if;
   					end_if;
   					if NOT EquipmentModules[i].0 then wrk_Aborting_to_Aborted:=(1*2**i)+temp_sum; end_if; // module is not enabled. therfor state is always true.
   					temp_sum:=wrk_Aborting_to_Aborted;
   				end_for;
   				Sts_SC_Status:=wrk_Aborting_to_Aborted;
   				Wrk_EM_Aborting:=wrk_Aborting_to_Aborted;
   				temp_sum:=0;
   				for i := 0 to 31 do										// scan from 0 till max array size
   					if Processes[i].0 then									// check if EquipmentModule is selected
   						if Processes[i].8 then		// Feedback from equipmentmodule
   							wrk_Aborting_to_Aborted:=(1*2**i)+temp_sum; 			// convert binary to dec value. sum= bits *2 ^ i. See https://flexiple.com/developers/decimal-to-binary-conversion
   					 	else
   							wrk_Aborting_to_Aborted:=(0*2**i)+temp_sum; 			// convert binary to dec value. sum= bits *2 ^ i. See https://flexiple.com/developers/decimal-to-binary-conversion
   						end_if;
   					end_if;
   					if NOT Processes[i].0 then wrk_Aborting_to_Aborted:=(1*2**i)+temp_sum; end_if; // module is not enabled. therfor state is always true.
   					temp_sum:=wrk_Aborting_to_Aborted;
   				end_for;
   				Wrk_Process_Aborting:=wrk_Aborting_to_Aborted;
   
   				if (Wrk_EM_Aborting = wrk_compare_UDINT) AND (Wrk_Process_Aborting = wrk_compare_UDINT)  then
   					MachineState:=9;												// move unit to aborted.
   				end_if;
   			else
   				MachineState:=9;
   			end_if;
   			#endregion
   
   
   
   		9:	/******************************************************		Aborted		******************************************************/
   			wrk_Aborting_to_Aborted	:=0; 											// clear old mem, since state was succesful.
   
   
   			if PackTags.Command.CntrlCmd = 9 AND PackTags.Command.CmdChangeRequest then	//	The tag holds the value of the command that provides the state command to drive a state change in the Base State Model
   				PackTags.Status.StateRequested:=1;									// request Aborted state.
   				MachineState:=1;													// move to clearing
   				PackTags.Command.CmdChangeRequest:=0;								//  accept request and set signal back low.
   			end_if;
   
   
   
   		10:	/******************************************************		Holding		******************************************************/
   			#region Check EquipmentModule StateControl (SC)
   			temp_sum:=0;
   
   			PackTags.Status.StateRequested:=11;										// request Held state.
   			if Cnf_EnableMachineStates.Holding then
   				for i := 0 to 31 do										// scan from 0 till max array size
   					if EquipmentModules[i].0 then									// check if EquipmentModule is selected
   						if EquipmentModules[i].10 then			// Feedback from equipmentmodule
   							wrk_Holding_to_Held:=(1*2**i)+temp_sum; 				// convert binary to dec value. sum= bits *2 ^ i. See https://flexiple.com/developers/decimal-to-binary-conversion
   					 	else
   							wrk_Holding_to_Held:=(0*2**i)+temp_sum; 				// convert binary to dec value. sum= bits *2 ^ i. See https://flexiple.com/developers/decimal-to-binary-conversion
   						end_if;
   					end_if;
   					if NOT EquipmentModules[i].0 then wrk_Holding_to_Held:=(1*2**i)+temp_sum; end_if; // module is not enabled. therfor state is always true.
   					temp_sum:=wrk_Holding_to_Held;
   				end_for;
   				Sts_SC_Status:=wrk_Holding_to_Held;
   				Wrk_EM_Holding:=wrk_Holding_to_Held;
   
   				temp_sum:=0;
   				for i := 0 to 31 do										// scan from 0 till max array size
   					if Processes[i].0 then									// check if EquipmentModule is selected
   						if Processes[i].10 then			// Feedback from equipmentmodule
   							wrk_Holding_to_Held:=(1*2**i)+temp_sum; 				// convert binary to dec value. sum= bits *2 ^ i. See https://flexiple.com/developers/decimal-to-binary-conversion
   					 	else
   							wrk_Holding_to_Held:=(0*2**i)+temp_sum; 				// convert binary to dec value. sum= bits *2 ^ i. See https://flexiple.com/developers/decimal-to-binary-conversion
   						end_if;
   					end_if;
   					if NOT Processes[i].0 then wrk_Holding_to_Held:=(1*2**i)+temp_sum; end_if; // module is not enabled. therfor state is always true.
   					temp_sum:=wrk_Holding_to_Held;
   				end_for;
   				Wrk_processes_Holding:=wrk_Holding_to_Held;
   
   				if (wrk_Holding_to_Held = wrk_compare_UDINT) AND (Wrk_processes_Holding = wrk_compare_UDINT) then
   					MachineState:=11;												// move unit to Held.
   				end_if;
   			else
   				MachineState:=11;
   			end_if;
   			#endregion
   
   
   
   		11:	/******************************************************		Held		******************************************************/
   			wrk_Holding_to_Held	:=0; 												// clear old mem, since state was succesful.
   
   			if Cnf_EnableMachineStates.Held then
   				if PackTags.Command.CntrlCmd = 5 AND PackTags.Command.CmdChangeRequest then	//	The tag holds the value of the command that provides the state command to drive a state change in the Base State Model
   					PackTags.Status.StateRequested:=12;									// request Unholding state.
   					MachineState:=12;													// move to unholding
   					PackTags.Command.CmdChangeRequest:=0;								//  accept request and set signal back low.
   				end_if;
   			else
   				PackTags.Status.StateRequested:=12;
   				MachineState:=12;
   				PackTags.Command.CmdChangeRequest:=0;
   			end_if;
   
   
   		12:	/******************************************************		Unholding	******************************************************/
   			#region Check EquipmentModule StateControl (SC)
   			temp_sum:=0;
   
   			PackTags.Status.StateRequested:=6;										// request Execute state.
   			if Cnf_EnableMachineStates.Unholding then
   				for i := 0 to 31 do										// scan from 0 till max array size
   					if EquipmentModules[i].0 then									// check if EquipmentModule is selected
   						if EquipmentModules[i].12 then		// Feedback from equipmentmodule
   							wrk_Unholding_to_Execute:=(1*2**i)+temp_sum; 			// convert binary to dec value. sum= bits *2 ^ i. See https://flexiple.com/developers/decimal-to-binary-conversion
   					 	else
   							wrk_Unholding_to_Execute:=(0*2**i)+temp_sum; 			// convert binary to dec value. sum= bits *2 ^ i. See https://flexiple.com/developers/decimal-to-binary-conversion
   						end_if;
   					end_if;
   					if NOT EquipmentModules[i].0 then wrk_Unholding_to_Execute:=(1*2**i)+temp_sum; end_if; // module is not enabled. therfor state is always true.
   					temp_sum:=wrk_Unholding_to_Execute;
   				end_for;
   				Sts_SC_Status:=wrk_Unholding_to_Execute;
   				Wrk_EM_Unholding:=wrk_Unholding_to_Execute;
   
   				temp_sum:=0;
   				for i := 0 to 31 do										// scan from 0 till max array size
   					if Processes[i].0 then									// check if EquipmentModule is selected
   						if Processes[i].12 then		// Feedback from equipmentmodule
   							wrk_Unholding_to_Execute:=(1*2**i)+temp_sum; 			// convert binary to dec value. sum= bits *2 ^ i. See https://flexiple.com/developers/decimal-to-binary-conversion
   					 	else
   							wrk_Unholding_to_Execute:=(0*2**i)+temp_sum; 			// convert binary to dec value. sum= bits *2 ^ i. See https://flexiple.com/developers/decimal-to-binary-conversion
   						end_if;
   					end_if;
   					if NOT Processes[i].0 then wrk_Unholding_to_Execute:=(1*2**i)+temp_sum; end_if; // module is not enabled. therfor state is always true.
   					temp_sum:=wrk_Unholding_to_Execute;
   				end_for;
   				Wrk_processes_Unholding:=wrk_Unholding_to_Execute;
   
   				if (wrk_Unholding_to_Execute = wrk_compare_UDINT) AND (Wrk_processes_Unholding = wrk_compare_UDINT) then
   					MachineState:=6;												// move unit to Execute.
   				end_if;
   			else
   				MachineState:=6;												// move unit to Execute.
   			end_if;
   			#endregion
   
   
   
   		13:	/******************************************************		Suspending	******************************************************/
   			#region Check EquipmentModule StateControl (SC)
   			temp_sum:=0;
   
   			PackTags.Status.StateRequested:=5;										// request Suspend state.
   			if Cnf_EnableMachineStates.Suspending then
   				for i := 0 to 31 do										// scan from 0 till max array size
   					if EquipmentModules[i].0 then									// check if EquipmentModule is selected
   						if EquipmentModules[i].13 then	// Feedback from equipmentmodule
   							wrk_Suspending_to_Suspended:=(1*2**i)+temp_sum; 		// convert binary to dec value. sum= bits *2 ^ i. See https://flexiple.com/developers/decimal-to-binary-conversion
   					 	else
   							wrk_Suspending_to_Suspended:=(0*2**i)+temp_sum; 		// convert binary to dec value. sum= bits *2 ^ i. See https://flexiple.com/developers/decimal-to-binary-conversion
   						end_if;
   					end_if;
   					if NOT EquipmentModules[i].0 then wrk_Suspending_to_Suspended:=(1*2**i)+temp_sum; end_if; // module is not enabled. therfor state is always true.
   					temp_sum:=wrk_Suspending_to_Suspended;
   				end_for;
   				Sts_SC_Status:=wrk_Suspending_to_Suspended;
   				Wrk_EM_Suspending:=wrk_Suspending_to_Suspended;
   
   				temp_sum:=0;
   				for i := 0 to 31 do										// scan from 0 till max array size
   					if Processes[i].0 then									// check if EquipmentModule is selected
   						if Processes[i].13 then	// Feedback from equipmentmodule
   							wrk_Suspending_to_Suspended:=(1*2**i)+temp_sum; 		// convert binary to dec value. sum= bits *2 ^ i. See https://flexiple.com/developers/decimal-to-binary-conversion
   					 	else
   							wrk_Suspending_to_Suspended:=(0*2**i)+temp_sum; 		// convert binary to dec value. sum= bits *2 ^ i. See https://flexiple.com/developers/decimal-to-binary-conversion
   						end_if;
   					end_if;
   					if NOT Processes[i].0 then wrk_Suspending_to_Suspended:=(1*2**i)+temp_sum; end_if; // module is not enabled. therfor state is always true.
   					temp_sum:=wrk_Suspending_to_Suspended;
   				end_for;
   				Wrk_processes_Suspending:=wrk_Suspending_to_Suspended;
   
   
   				if (Wrk_EM_Suspending = wrk_compare_UDINT) AND (Wrk_processes_Suspending = wrk_compare_UDINT) then
   					MachineState:=5;												// move unit to Suspend.
   				end_if;
   			else
   				MachineState:=5;												// move unit to Suspend.
   			end_if;
   			#endregion
   
   
   
   		14:	/******************************************************		Unsuspending ******************************************************/
   			#region Check EquipmentModule StateControl (SC)
   			temp_sum:=0;
   
   			PackTags.Status.StateRequested:=6;										// request Execute state.
   			if Cnf_EnableMachineStates.Unsuspending then
   				for i := 0 to 31 do										// scan from 0 till max array size
   					if EquipmentModules[i].0 then									// check if EquipmentModule is selected
   						if EquipmentModules[i].14 then	// Feedback from equipmentmodule
   							wrk_Unsuspending_to_Execute:=(1*2**i)+temp_sum; 		// convert binary to dec value. sum= bits *2 ^ i. See https://flexiple.com/developers/decimal-to-binary-conversion
   					 	else
   							wrk_Unsuspending_to_Execute:=(0*2**i)+temp_sum; 		// convert binary to dec value. sum= bits *2 ^ i. See https://flexiple.com/developers/decimal-to-binary-conversion
   						end_if;
   					end_if;
   					if NOT EquipmentModules[i].0 then wrk_Unsuspending_to_Execute:=(1*2**i)+temp_sum; end_if; // module is not enabled. therfor state is always true.
   					temp_sum:=wrk_Unsuspending_to_Execute;
   				end_for;
   				Sts_SC_Status:=wrk_Unsuspending_to_Execute;
   				Wrk_EM_Unsuspending:=wrk_Unsuspending_to_Execute;
   
   				temp_sum:=0;
   				for i := 0 to 31 do										// scan from 0 till max array size
   					if Processes[i].0 then									// check if EquipmentModule is selected
   						if Processes[i].14 then	// Feedback from equipmentmodule
   							wrk_Unsuspending_to_Execute:=(1*2**i)+temp_sum; 		// convert binary to dec value. sum= bits *2 ^ i. See https://flexiple.com/developers/decimal-to-binary-conversion
   					 	else
   							wrk_Unsuspending_to_Execute:=(0*2**i)+temp_sum; 		// convert binary to dec value. sum= bits *2 ^ i. See https://flexiple.com/developers/decimal-to-binary-conversion
   						end_if;
   					end_if;
   					if NOT Processes[i].0 then wrk_Unsuspending_to_Execute:=(1*2**i)+temp_sum; end_if; // module is not enabled. therfor state is always true.
   					temp_sum:=wrk_Unsuspending_to_Execute;
   				end_for;
   				Wrk_processes_Unsuspending:=wrk_Unsuspending_to_Execute;
   
   				if (Wrk_EM_Unsuspending = wrk_compare_UDINT) AND (Wrk_processes_Unsuspending = wrk_compare_UDINT) then
   					MachineState:=6;													// move unit to Execute.
   				end_if;
   			else
   				MachineState:=6;													// move unit to Execute.
   			end_if;
   			#endregion
   
   
   
   		15:	/******************************************************		Resetting	******************************************************/
   			#region Check EquipmentModule StateControl (SC)
   			temp_sum:=0;
   			PackTags.Status.StateRequested:=4;										// request Idle state.
   			wrk_HandHalt:=0;
   			if Cnf_EnableMachineStates.Resetting then
   				if T_ResetSignal_OFF.DN then											// wait for reset seq for unit
   					for i := 0 to 31 do										// scan from 0 till max array size
   						if EquipmentModules[i].0 then									// check if EquipmentModule is selected
   							if EquipmentModules[i].15 then			// Feedback from equipmentmodule
   								wrk_Resetting_to_Idle:=(1*2**i)+temp_sum; 				// convert binary to dec value. sum= bits *2 ^ i. See https://flexiple.com/developers/decimal-to-binary-conversion
   						 	else
   								wrk_Resetting_to_Idle:=(0*2**i)+temp_sum; 				// convert binary to dec value. sum= bits *2 ^ i. See https://flexiple.com/developers/decimal-to-binary-conversion
   							end_if;
   						end_if;
   						if NOT EquipmentModules[i].0 then wrk_Resetting_to_Idle:=(1*2**i)+temp_sum; end_if; // module is not enabled. therfor state is always true.
   						temp_sum:=wrk_Resetting_to_Idle;
   					end_for;
   					Wrk_EM_Restting:=wrk_Resetting_to_Idle;
   					Sts_SC_Status:=wrk_Resetting_to_Idle;
   
   					temp_sum:=0;
   					for i := 0 to 31 do										// scan from 0 till max array size
   						if Processes[i].0 then									// check if EquipmentModule is selected
   							if Processes[i].15 then			// Feedback from equipmentmodule
   								wrk_Resetting_to_Idle:=(1*2**i)+temp_sum; 				// convert binary to dec value. sum= bits *2 ^ i. See https://flexiple.com/developers/decimal-to-binary-conversion
   						 	else
   								wrk_Resetting_to_Idle:=(0*2**i)+temp_sum; 				// convert binary to dec value. sum= bits *2 ^ i. See https://flexiple.com/developers/decimal-to-binary-conversion
   							end_if;
   						end_if;
   						if NOT Processes[i].0 then wrk_Resetting_to_Idle:=(1*2**i)+temp_sum; end_if; // module is not enabled. therfor state is always true.
   						temp_sum:=wrk_Resetting_to_Idle;
   					end_for;
   					Wrk_Process_Restting:=wrk_Resetting_to_Idle;
   
   
   					if (Wrk_EM_Restting = wrk_compare_UDINT) AND (Wrk_Process_Restting = wrk_compare_UDINT) then
   						MachineState:=4;												// move unit to Idle.
   					end_if;
   				end_if;
   			else
   				MachineState:=4;												// move unit to Idle.
   			end_if;
   			#endregion
   
   
   
   		16:	/******************************************************		Completing	******************************************************/
   			#region Check EquipmentModule StateControl (SC)
   			temp_sum:=0;
   
   			PackTags.Status.StateRequested:=17;										// request Complete state.
   			if Cnf_EnableMachineStates.Completing then
   				for i := 0 to 31 do										// scan from 0 till max array size
   					if EquipmentModules[i].0 then									// check if EquipmentModule is selected
   						if EquipmentModules[i].16 then	// Feedback from equipmentmodule
   							wrk_Completing_to_Completed:=(1*2**i)+temp_sum; 		// convert binary to dec value. sum= bits *2 ^ i. See https://flexiple.com/developers/decimal-to-binary-conversion
   					 	else
   							wrk_Completing_to_Completed:=(0*2**i)+temp_sum; 		// convert binary to dec value. sum= bits *2 ^ i. See https://flexiple.com/developers/decimal-to-binary-conversion
   						end_if;
   					end_if;
   					if NOT EquipmentModules[i].0 then wrk_Completing_to_Completed:=(1*2**i)+temp_sum; end_if; // module is not enabled. therfor state is always true.
   					temp_sum:=wrk_Completing_to_Completed;
   				end_for;
   				Sts_SC_Status:=wrk_Completing_to_Completed;
   				Wrk_EM_Completed:=wrk_Completing_to_Completed;
   
   				temp_sum:=0;
   				for i := 0 to 31 do										// scan from 0 till max array size
   					if Processes[i].0 then									// check if EquipmentModule is selected
   						if Processes[i].16 then	// Feedback from equipmentmodule
   							wrk_Completing_to_Completed:=(1*2**i)+temp_sum; 		// convert binary to dec value. sum= bits *2 ^ i. See https://flexiple.com/developers/decimal-to-binary-conversion
   					 	else
   							wrk_Completing_to_Completed:=(0*2**i)+temp_sum; 		// convert binary to dec value. sum= bits *2 ^ i. See https://flexiple.com/developers/decimal-to-binary-conversion
   						end_if;
   					end_if;
   					if NOT Processes[i].0 then wrk_Completing_to_Completed:=(1*2**i)+temp_sum; end_if; // module is not enabled. therfor state is always true.
   					temp_sum:=wrk_Completing_to_Completed;
   				end_for;
   				Wrk_processes_Completed:=wrk_Completing_to_Completed;
   
   
   
   				if (Wrk_EM_Completed = wrk_compare_UDINT) AND (Wrk_processes_Completed = wrk_compare_UDINT) then
   					MachineState:=17;												// move unit to Complete.
   				end_if;
   			else
   				MachineState:=17;												// move unit to Complete.
   			end_if;
   			#endregion
   
   
   
   		17:	/******************************************************		Complete	******************************************************/
   			wrk_Completing_to_Completed	:=0; 										// clear old mem, since state was succesful.
   
   			if Cnf_EnableMachineStates.Complete then
   				if PackTags.Command.CntrlCmd = 1 AND PackTags.Command.CmdChangeRequest then	//	The tag holds the value of the command that provides the state command to drive a state change in the Base State Model
   					PackTags.Status.StateRequested:=15;									// request Resetting state.
   					MachineState:=15;													// move to resetting
   					PackTags.Command.CmdChangeRequest:=0;								//  accept request and set signal back low.
   				end_if;
   			else
   				PackTags.Status.StateRequested:=15;									// request Resetting state.
   				MachineState:=15;													// move to resetting
   				PackTags.Command.CmdChangeRequest:=0;								//  accept request and set signal back low.
   			end_if;
   
   
   		/**************************************************************************************************************************************/
   		else
   		MachineState:=8;	// MachineState is undefined, forces machine to state aborting. Equipment reacts accordingly.
   	end_case;
   	#region Recieve command(alarm,Fault,Suspend)
   		for i := 0 to 31 do
   
   			if NOT (Sts_Aborting OR Sts_Aborted OR Sts_Clearing OR Sts_Stopping OR Sts_Stopped) Then
   				if EquipmentModules[i].0 AND EquipmentModules[i].22 AND NOT Sts_MachineFaulted then
   					Sts_MachineFaulted				:=TRUE;								// Set machine faulted to true.
   					PackTags.Status.StateRequested	:=7;								// request Stopping state.
   					MachineState					:=7;								// move to Stopping
   				end_if;
   			end_if;
   			if NOT (Sts_Aborting OR Sts_Aborted OR Sts_Clearing OR Sts_Stopping OR Sts_Stopped) Then
   				if Processes[i].0 AND Processes[i].22 AND NOT Sts_MachineFaulted then
   					Sts_MachineFaulted				:=TRUE;								// Set machine faulted to true.
   					PackTags.Status.StateRequested	:=7;								// request Stopping state.
   					MachineState					:=7;								// move to Stopping
   				end_if;
   			end_if;
   
   			if EquipmentModules[i].0 AND EquipmentModules[i].23 AND NOT Sts_MachineFaulted then
   				Sts_MachineFaulted				:=TRUE;								// Set machine faulted to true.
   				PackTags.Status.StateRequested	:=8;								// request Aborting state.
   				MachineState					:=8;								// move to aborting
   			end_if;
   			if Processes[i].0 AND Processes[i].23 AND NOT Sts_MachineFaulted then
   				Sts_MachineFaulted				:=TRUE;								// Set machine faulted to true.
   				PackTags.Status.StateRequested	:=8;								// request Aborting state.
   				MachineState					:=8;								// move to aborting
   			end_if;
   
   			if Sts_Execute then
   				if EquipmentModules[i].0 AND EquipmentModules[i].20 AND NOT (Sts_Suspended OR Sts_Suspending)  then
   					PackTags.Status.StateRequested	:=13;								// request Aborting state.
   					MachineState					:=13;								// move to aborting
   				end_if;
   				if Processes[i].0 AND Processes[i].20 AND NOT (Sts_Suspended OR Sts_Suspending)  then
   					PackTags.Status.StateRequested	:=13;								// request Aborting state.
   					MachineState					:=13;								// move to aborting
   				end_if;
   			end_if;
   		end_for;
   	#endregion
   	#region HMI stop / abort command
   	/*
   	User should always be able to stop / abort the machine. however this is there is some logic regarding the stop & abort.
   	if the machine is in aborting the user can not give a stop trigger and bypass aborted / clearing.
   	*/
   
   		/* Stopping command */
   		if (PackTags.Command.CntrlCmd = 3 AND PackTags.Command.CmdChangeRequest) AND NOT (Sts_Aborted OR Sts_Aborting OR Sts_Stopping OR Sts_Clearing) then
   				wrk_HandHalt					:=1;								// User forced machine to stop state.
   				PackTags.Command.CmdChangeRequest:=0;
   				PackTags.Status.StateRequested	:=7;								// request Stopping state.
   				MachineState					:=7;								// move to Stopping
   		end_if;
   
   		/* Aborting command	*/
   		if (PackTags.Command.CntrlCmd = 8 AND PackTags.Command.CmdChangeRequest) AND NOT (Sts_Aborting) then
   				wrk_HandHalt					:=1;								// User forced machine to abort state.
   				PackTags.Command.CmdChangeRequest:=0;
   				PackTags.Status.StateRequested	:=8;								// request Aborting state.
   				MachineState					:=8;								// move to aborting
   		end_if;
   	#endregion
   #endregion
   #region Feedback to user
   	PackTags.Status.UnitFaulted:=Sts_MachineFaulted;								// machine fualted to packtag
   	if PackTags.Status.StateRequested <> PackTags.Status.StateCurrent then			// compare current state with requested state done above.
   		PackTags.Status.StateChangeInProcess:=TRUE;									// State trans is active.
   	else
   		PackTags.Status.StateChangeInProcess:=FALSE;								// State trans is NOT active.
   	end_if;
   	if (wrk_prev_state<>MachineState) OR S:fs then
   		Sts_Clearing	:=	FALSE;					// clear old mem
   		Sts_Stopped		:=	FALSE;					// clear old mem
   		Sts_Starting	:=	FALSE;					// clear old mem
   		Sts_Idle		:=	FALSE;					// clear old mem
   		Sts_Suspended	:=	FALSE;					// clear old mem
   		Sts_Execute		:=	FALSE;					// clear old mem
   		Sts_Stopping	:=	FALSE;					// clear old mem
   		Sts_Aborting	:=	FALSE;					// clear old mem
   		Sts_Aborted		:=	FALSE;					// clear old mem
   		Sts_Holding		:=	FALSE;					// clear old mem
   		Sts_Held		:=	FALSE;					// clear old mem
   		Sts_Unholding	:=	FALSE;					// clear old mem
   		Sts_Suspending	:=	FALSE;					// clear old mem
   		Sts_Unsuspending:=	FALSE;					// clear old mem
   		Sts_Resetting	:=	FALSE;					// clear old mem
   		Sts_Completing	:=	FALSE;					// clear old mem
   		Sts_Complete	:=	FALSE;					// clear old mem
   		case MachineState of						// Case handler
   			1: 	Sts_Clearing	:=	TRUE;			// state is true.
   			2: 	Sts_Stopped		:=	TRUE;			// state is true.
   			3: 	Sts_Starting	:=	TRUE;			// state is true.
   			4: 	Sts_Idle		:=	TRUE;			// state is true.
   			5: 	Sts_Suspended	:=	TRUE;			// state is true.
   			6: 	Sts_Execute		:=	TRUE;			// state is true.
   			7: 	Sts_Stopping	:=	TRUE;			// state is true.
   			8: 	Sts_Aborting	:=	TRUE;			// state is true.
   			9: 	Sts_Aborted		:=	TRUE;			// state is true.
   			10: Sts_Holding		:=	TRUE;			// state is true.
   			11:	Sts_Held		:=	TRUE;			// state is true.
   			12:	Sts_Unholding	:=	TRUE;			// state is true.
   			13:	Sts_Suspending	:=	TRUE;			// state is true.
   			14:	Sts_Unsuspending:=	TRUE;			// state is true.
   			15:	Sts_Resetting	:=	TRUE;			// state is true.
   			16:	Sts_Completing	:=	TRUE;			// state is true.
   			17:	Sts_Complete	:=	TRUE;			// state is true.
   			else
   			wrk_prev_state	:=	MachineState;		// undefined state.
   		end_case;
   		wrk_prev_state	:=	MachineState;			// Finish while loop by setting machinestate to previous state.
   	end_if;
   	PackTags.Status.StateCurrent:=MachineState;		// current state is shown as copy of MachineState local. since Case is using same numric as StateCurrent according to TR88_0002
   #endregion
   #region Administration Tags
   	#region ModeCurrentTime
   		if T_second_puls.DN then
   			case MachineMode of																//	Case handler
   				1: PackTags.Admin.ModeCurrentTime[1]:=PackTags.Admin.ModeCurrentTime[1]+1; 		//	Production count
   				2: PackTags.Admin.ModeCurrentTime[2]:=PackTags.Admin.ModeCurrentTime[2]+1; 		//	Maintenance count
   				3: PackTags.Admin.ModeCurrentTime[3]:=PackTags.Admin.ModeCurrentTime[3]+1; 		//	Manual count
   				else
   				// undefined state
   			end_case;
   			if MachineMode <> 1 then PackTags.Admin.ModeCurrentTime[1]:=0; end_if; 			//	if machine is not in this state, reset count
   			if MachineMode <> 2 then PackTags.Admin.ModeCurrentTime[2]:=0; end_if; 			//	if machine is not in this state, reset count
   			if MachineMode <> 3 then PackTags.Admin.ModeCurrentTime[3]:=0; end_if; 			//	if machine is not in this state, reset count
   
   		end_if;
   	#endregion
   
   
   	#region ModeCumulativeTime
   		if T_second_puls.DN then
   			case MachineMode of																		//	Case handler
   				1: PackTags.Admin.ModeCumulativeTime[1]:=PackTags.Admin.ModeCumulativeTime[1]+1; 		//	Production count
   				2: PackTags.Admin.ModeCumulativeTime[2]:=PackTags.Admin.ModeCumulativeTime[2]+1; 		//	Maintenance count
   				3: PackTags.Admin.ModeCumulativeTime[3]:=PackTags.Admin.ModeCumulativeTime[3]+1; 		//	Manual count
   				else
   				// undefined state
   			end_case;
   		end_if;
   	#endregion
   
   	#region StateCurrentTime[Mode,State]
   		if T_second_puls.DN then
   			for i := 0 to 3 do
   				for k := 0 to 17 do
   					if (i = MachineMode) AND (k=MachineState) then
   						// do nothing since this is the current state.
   					else
   						PackTags.Admin.StateCurrentTime[i].Mode[k]:=0;	// reset time value
   					end_if;
   				end_for;
   			end_for;
   			case MachineState of						// Case handler
   				1:  PackTags.Admin.StateCurrentTime[MachineMode].Mode[1]	:=	PackTags.Admin.StateCurrentTime[MachineMode].Mode[1]+1;
   				2:  PackTags.Admin.StateCurrentTime[MachineMode].Mode[2]	:=	PackTags.Admin.StateCurrentTime[MachineMode].Mode[2]+1;
   				3:  PackTags.Admin.StateCurrentTime[MachineMode].Mode[3]	:=	PackTags.Admin.StateCurrentTime[MachineMode].Mode[3]+1;
   				4:  PackTags.Admin.StateCurrentTime[MachineMode].Mode[4]	:=	PackTags.Admin.StateCurrentTime[MachineMode].Mode[4]+1;
   				5:  PackTags.Admin.StateCurrentTime[MachineMode].Mode[5]	:=	PackTags.Admin.StateCurrentTime[MachineMode].Mode[5]+1;
   				6:  PackTags.Admin.StateCurrentTime[MachineMode].Mode[6]	:=	PackTags.Admin.StateCurrentTime[MachineMode].Mode[6]+1;
   				7:  PackTags.Admin.StateCurrentTime[MachineMode].Mode[7]	:=	PackTags.Admin.StateCurrentTime[MachineMode].Mode[7]+1;
   				8:  PackTags.Admin.StateCurrentTime[MachineMode].Mode[8]	:=	PackTags.Admin.StateCurrentTime[MachineMode].Mode[8]+1;
   				9:  PackTags.Admin.StateCurrentTime[MachineMode].Mode[9]	:=	PackTags.Admin.StateCurrentTime[MachineMode].Mode[9]+1;
   				10: PackTags.Admin.StateCurrentTime[MachineMode].Mode[10]	:=	PackTags.Admin.StateCurrentTime[MachineMode].Mode[10]+1;
   				11:	PackTags.Admin.StateCurrentTime[MachineMode].Mode[11]	:=	PackTags.Admin.StateCurrentTime[MachineMode].Mode[11]+1;
   				12:	PackTags.Admin.StateCurrentTime[MachineMode].Mode[12]	:=	PackTags.Admin.StateCurrentTime[MachineMode].Mode[12]+1;
   				13:	PackTags.Admin.StateCurrentTime[MachineMode].Mode[13]	:=	PackTags.Admin.StateCurrentTime[MachineMode].Mode[13]+1;
   				14:	PackTags.Admin.StateCurrentTime[MachineMode].Mode[14]	:=	PackTags.Admin.StateCurrentTime[MachineMode].Mode[14]+1;
   				15:	PackTags.Admin.StateCurrentTime[MachineMode].Mode[15]	:=	PackTags.Admin.StateCurrentTime[MachineMode].Mode[15]+1;
   				16:	PackTags.Admin.StateCurrentTime[MachineMode].Mode[16]	:=	PackTags.Admin.StateCurrentTime[MachineMode].Mode[16]+1;
   				17:	PackTags.Admin.StateCurrentTime[MachineMode].Mode[17]	:=	PackTags.Admin.StateCurrentTime[MachineMode].Mode[17]+1;
   				else
   				// undefined state.
   			end_case;
   		end_if;
   	#endregion
   
   	#region StateCumulativeTime[Mode,State]
   		if T_second_puls.DN then
   			case MachineState of						// Case handler
   				1:  PackTags.Admin.StateCumulativeTime[MachineMode].Mode[1]		:=	PackTags.Admin.StateCumulativeTime[MachineMode].Mode[1]+1;
   				2:  PackTags.Admin.StateCumulativeTime[MachineMode].Mode[2]		:=	PackTags.Admin.StateCumulativeTime[MachineMode].Mode[2]+1;
   				3:  PackTags.Admin.StateCumulativeTime[MachineMode].Mode[3]		:=	PackTags.Admin.StateCumulativeTime[MachineMode].Mode[3]+1;
   				4:  PackTags.Admin.StateCumulativeTime[MachineMode].Mode[4]		:=	PackTags.Admin.StateCumulativeTime[MachineMode].Mode[4]+1;
   				5:  PackTags.Admin.StateCumulativeTime[MachineMode].Mode[5]		:=	PackTags.Admin.StateCumulativeTime[MachineMode].Mode[5]+1;
   				6:  PackTags.Admin.StateCumulativeTime[MachineMode].Mode[6]		:=	PackTags.Admin.StateCumulativeTime[MachineMode].Mode[6]+1;
   				7:  PackTags.Admin.StateCumulativeTime[MachineMode].Mode[7]		:=	PackTags.Admin.StateCumulativeTime[MachineMode].Mode[7]+1;
   				8:  PackTags.Admin.StateCumulativeTime[MachineMode].Mode[8]		:=	PackTags.Admin.StateCumulativeTime[MachineMode].Mode[8]+1;
   				9:  PackTags.Admin.StateCumulativeTime[MachineMode].Mode[9]		:=	PackTags.Admin.StateCumulativeTime[MachineMode].Mode[9]+1;
   				10: PackTags.Admin.StateCumulativeTime[MachineMode].Mode[10]	:=	PackTags.Admin.StateCumulativeTime[MachineMode].Mode[10]+1;
   				11:	PackTags.Admin.StateCumulativeTime[MachineMode].Mode[11]	:=	PackTags.Admin.StateCumulativeTime[MachineMode].Mode[11]+1;
   				12:	PackTags.Admin.StateCumulativeTime[MachineMode].Mode[12]	:=	PackTags.Admin.StateCumulativeTime[MachineMode].Mode[12]+1;
   				13:	PackTags.Admin.StateCumulativeTime[MachineMode].Mode[13]	:=	PackTags.Admin.StateCumulativeTime[MachineMode].Mode[13]+1;
   				14:	PackTags.Admin.StateCumulativeTime[MachineMode].Mode[14]	:=	PackTags.Admin.StateCumulativeTime[MachineMode].Mode[14]+1;
   				15:	PackTags.Admin.StateCumulativeTime[MachineMode].Mode[15]	:=	PackTags.Admin.StateCumulativeTime[MachineMode].Mode[15]+1;
   				16:	PackTags.Admin.StateCumulativeTime[MachineMode].Mode[16]	:=	PackTags.Admin.StateCumulativeTime[MachineMode].Mode[16]+1;
   				17:	PackTags.Admin.StateCumulativeTime[MachineMode].Mode[17]	:=	PackTags.Admin.StateCumulativeTime[MachineMode].Mode[17]+1;
   				else
   				// undefined state.
   			end_case;
   		end_if;
   
   	#endregion
   
   	#region AccTimeSinceReset
   		if T_second_puls.DN then
   			if NOT Sts_Resetting then PackTags.Admin.AccTimeSinceReset:=PackTags.Admin.AccTimeSinceReset+1; end_if;		// count until machine has been in resetting.
   		end_if;
   		if T_ResetSignal_ON.TT OR T_ResetSignal_HMI.TT then PackTags.Admin.AccTimeSinceReset:=0; end_if;
   	#endregion
   
   	#region PACDateTime
   	GSV(WallClockTime,,CurrentValue,wrk_DateTime);
   		#region PACDateTime.Date
   			PackTags.Admin.PACDateTime.Date:=wrk_DateTime;
   		#endregion
   		#region PACDateTime.Time
   			PackTags.Admin.PACDateTime.Time:=wrk_DateTime;
   		#endregion
   	#endregion
   #endregion
   #region HMI data representation
   	if StateHistory[0].State_Num <> MachineState then
   		for i := 1 to 9 do
   			StateHistory[10-i].State_Num 			:= StateHistory[9-i].State_Num;
   			StateHistory[10-i].Time_Spend_in_State 	:= StateHistory[9-i].Time_Spend_in_State;
   			StateHistory[10-i].Time_enteringState 	:= StateHistory[9-i].Time_enteringState;
   		end_for;
   		StateHistory[0].State_Num			:=MachineState;
   		StateHistory[0].Time_enteringState	:=wrk_DateTime;
   	end_if;
   	StateHistory[0].Time_Spend_in_State	:=PackTags.Admin.StateCurrentTime[MachineMode].Mode[MachineState];
   #endregion
END_ROUTINE
